// TIA Portal V20 export
VAR_GLOBAL   // PLC tag table "Unit1Em4_Servo"
   "BA030AZSBK04.04" AT %I1012.4 : Bool;   // ANODE MAIN P&P2 LIMITS SENSOR(-)
   "BA030AZSBK04.05" AT %I1012.5 : Bool;   // ANODE MAIN P&P2 LIMITS SENSOR(+)
   "BA030AZSBK04.14" AT %I1013.4 : Bool;   // ANODE MAIN P&P2 LIMITS SENSOR HOME
   "BA030AZSBK05.00" AT %I1016.0 : Bool;   // ANODE MAIN P&P1 Z-AXIS LIMIT SENSOR(-)
   "BA030AZSBK05.01" AT %I1016.1 : Bool;   // ANODE MAIN P&P1 Z-AXIS LIMIT SENSOR(+)
   "BA030AZSBK05.02" AT %I1016.2 : Bool;   // ANODE MAIN P&P1 Y-AXIS LIMIT SENSOR(-)
   "BA030AZSBK05.03" AT %I1016.3 : Bool;   // ANODE MAIN P&P1 Y-AXIS LIMIT SENSOR(+)
   "BA030AZSBK05.10" AT %I1017.0 : Bool;   // ANODE MAIN P&P1 Z-AXIS HOME SENSOR
   "BA030AZSBK05.12" AT %I1017.2 : Bool;   // ANODE MAIN P&P1 Y-AXIS HOME SENSOR
   "BA030AZSBK06.00" AT %I1020.0 : Bool;   // ANODE MAIN P&P2 Z-AXIS LIMIT SENSOR(-)
   "BA030AZSBK06.01" AT %I1020.1 : Bool;   // ANODE MAIN P&P2 Z-AXIS HOME SENSOR
   "BA030AZSBK06.02" AT %I1020.2 : Bool;   // ANODE MAIN P&P2 Z-AXIS LIMIT SENSOR(+)
   "BA030AZSBK09.00" AT %I1032.0 : Bool;   // ANODE ALIGN TABLE X-AXIS LIMIT SENSOR(-)
   "BA030AZSBK09.01" AT %I1032.1 : Bool;   // ANODE ALIGN TABLE X-AXIS LIMIT SENSOR(+)
   "BA030AZSBK09.02" AT %I1032.2 : Bool;   // ANODE ALIGN TABLE Y1-AXIS LIMIT SENSOR(-)
   "BA030AZSBK09.03" AT %I1032.3 : Bool;   // ANODE ALIGN TABLE Y1-AXIS LIMIT SENSOR(+)
   "BA030AZSBK09.04" AT %I1032.4 : Bool;   // ANODE ALIGN TABLE Y2-AXIS LIMIT SENSOR(-)
   "BA030AZSBK09.05" AT %I1032.5 : Bool;   // ANODE ALIGN TABLE Y2-AXIS LIMIT SENSOR(+)
   "BA030AZSBK09.10" AT %I1033.0 : Bool;   // ANODE ALIGN TABLE X-AXIS HOME SENSOR
   "BA030AZSBK09.12" AT %I1033.2 : Bool;   // ANODE ALIGN TABLE Y1-AXIS HOME SENSOR
   "BA030AZSBK09.14" AT %I1033.4 : Bool;   // ANODE ALIGN TABLE Y2-AXIS HOME SENSOR
   "BA030AZSBK04.00" AT %I1012.0 : Bool;   // ANODE MAIN P&P1 X-AXIS LIMITS SENSOR(-)
   "BA030AZSBK04.01" AT %I1012.1 : Bool;   // ANODE MAIN P&P1 X-AXIS LIMITS SENSOR(+)
   "BA030AZSBK04.10" AT %I1013.0 : Bool;   // ANODE MAIN P&P1 X-AXIS LIMITS SENSOR HOME
END_VAR
